// TwinCAT 3 PLC project PLC1
// ProgramVersion: 3.1.4023.0
// libraries:
//   Tc2_Standard, * (Beckhoff Automation GmbH)
//   Tc2_System, * (Beckhoff Automation GmbH)
//   Tc2_Utilities, * (Beckhoff Automation GmbH)
//   Tc3_Database, * (Beckhoff Automation GmbH)
//   Tc3_EventLogger, * (Beckhoff Automation GmbH)
//   Tc3_JsonXml, * (Beckhoff Automation GmbH)
//   Tc3_Module, * (Beckhoff Automation GmbH)
// project tree:
//   / DBTask.TcTTO
//   DUTs/ stData.TcDUT
//   GVLs/ GlobalData.TcGVL
//   POUs/ GetLocalData.TcPOU, GetLocalPlcEx.TcPOU, PostRemoteData.TcPOU, UpdateSync.TcPOU
// real-time tasks:
//   TASK PlcTask: cycle T#1ms, priority 20, ADS port 350
//   TASK PlcUpdateData: cycle T#100us, priority 21, ADS port 351
//   TASK DBTask: cycle T#100us, priority 22, ADS port 352

CONFIGURATION PLC1
    RESOURCE PLC ON TwinCAT3
        TASK DBTask(INTERVAL := T#100us, PRIORITY := 22);
        PROGRAM GetLocalData WITH DBTask : GetLocalData;
        PROGRAM PostRemoteData WITH DBTask : PostRemoteData;
        PROGRAM UpdateSync WITH DBTask : UpdateSync;
    END_RESOURCE
END_CONFIGURATION

// ---- DUTs/stData.TcDUT
TYPE stData :
STRUCT
	iId: LINT;
	bSync: BOOL;
	dtTimestamp: DT;
	rSpeed: LREAL;
	rPos: LREAL;
	bPulse: BOOL;
END_STRUCT
END_TYPE

// ---- GVLs/GlobalData.TcGVL
{attribute 'qualified_only'}
VAR_GLOBAL
	bRemotePosted: BOOL := FALSE;
	bLocalGot: BOOL:= FALSE;
	blocalUpdated: BOOL:= TRUE;
	bMeasure: BOOL;
	aReadStruct : stData;
END_VAR

// ---- POUs/GetLocalData.TcPOU
PROGRAM GetLocalData
VAR
	fbSqlDatabase : FB_SQLDatabaseEvt(sNetID := '', tTimeout := T#5S);
	fbSqlCommand : FB_SQLCommandEvt(sNetID := '', tTimeout := T#5S);
	fbSqlResult: FB_SQLResultEvt(sNetID:='', tTimeout := T#5S);
	myDBID: UDINT := 1;
	sTableName: STRING := 'Data';
	sCmd: STRING(1000);

	tcMessage1 : I_TcMessage;
	tcMessage2 : I_TcMessage;
	tcMessage3 : I_TcMessage;
	tcMessage4 : I_TcMessage;

	systime: GETSYSTEMTIME;
	currentTime: T_FILETIME;
	iId: LINT := 1;
	
	bFirstScan: BOOL := TRUE;
	bExecute: bool;
	fbTon: TON;
	bLapse: BOOL := FALSE;
	bRead: BOOL:= FALSE;
	
	temp: INT;
END_VAR

IF (bFirstScan) THEN
	IF fbSqlDatabase.Connect(myDBID) THEN
		bFirstScan := FALSE;
		IF fbSqlDatabase.bError THEN
			tcMessage1:= fbSqlDatabase.ipTcResult;
			bFirstScan := TRUE;
		END_IF
	END_IF
END_IF

fbTon(IN:= NOT fbTon.Q, PT:= T#100mS);
IF fbTon.Q THEN
	bExecute := TRUE;
END_IF

IF bExecute AND NOT bFirstScan AND GlobalData.blocalUpdated THEN
	GlobalData.bMeasure:= TRUE;
	CreateSelect();
		
	IF fbSqlDatabase.CreateCmd(ADR(fbSqlCommand)) THEN
		IF fbSqlDatabase.bError THEN
			tcMessage2:= fbSqlDatabase.ipTcResult;
		END_IF
	END_IF
		
	IF NOT bRead THEN 
		IF fbSQLCommand.ExecuteDataReturn(ADR(sCmd), LEN(sCmd), ADR(fbSqlResult)) THEN
			IF fbSQLCommand.bError THEN
				tcMessage3 := fbSQLCommand.ipTcResult;
			END_IF
			bRead:= TRUE;
		END_IF
	ELSE
		IF fbSqlResult.Read(0, 1, ADR(GlobalData.aReadStruct), SIZEOF(GlobalData.aReadStruct), FALSE, TRUE) THEN
			IF fbSqlResult.bError THEN
				tcMessage4:= fbSqlResult.ipTcResult;
			END_IF
			bRead:= FALSE;
			bExecute:= FALSE;
			IF GlobalData.aReadStruct.iId <> 0 THEN
				GlobalData.blocalUpdated:= FALSE;
				GlobalData.bLocalGot:= TRUE;
			END_IF
		END_IF
	END_IF
	
END_IF

ACTION CreateSelect:
sCmd := 'SELECT * FROM ';
sCmd := concat(sCmd, sTableName);
sCmd := concat(sCmd, ' WHERE Sync=0 LIMIT 1');
END_ACTION

END_PROGRAM

// ---- POUs/PostRemoteData.TcPOU
PROGRAM PostRemoteData
VAR
	//Query Builder for Document DB
	fbNoSqlQueryBuilder_DocumentDB: FB_NoSQLQueryBuilder_DocumentDB;
	InsertQueryOption: T_QueryOptionDocumentDB_Insert;
	sDocument: STRING (1000);
	sDBName: STRING := 'Datalog';

	//Document json writer
	fbJsonWriter: FB_JsonSaxWriter;
	
	//Query Execution
	fbNoSqlQuery: FB_NoSQLQueryEvt(sNetID:= '', tTimeout:= T#5S);
	myDBID: UDINT := 2;
	TcMessage: I_TcMessage;
END_VAR

IF GlobalData.bLocalGot THEN
	CreateQuery();
	CreateDocument();
	
	IF fbNoSqlQuery.Execute(hDBID:= myDBID, iNoSQLQueryBuilder:= fbNoSqlQueryBuilder_DocumentDB) THEN
		GlobalData.bLocalGot := FALSE;
		GlobalData.bRemotePosted := TRUE;
		IF fbNoSqlQuery.bError THEN
			TcMessage:= fbNoSqlQuery.ipTcResult;
			GlobalData.bLocalGot := TRUE;
			GlobalData.bRemotePosted := FALSE;
		END_IF
	END_IF
END_IF

ACTION CreateDocument:
fbJsonWriter.StartObject();
fbJsonWriter.AddKey('Timestamp');
fbJsonWriter.AddDateTime(GlobalData.aReadStruct.dtTimestamp);
fbJsonWriter.AddKey('Speed');
fbJsonWriter.AddLreal(GlobalData.aReadStruct.rSpeed);
fbJsonWriter.AddKey('Pos');
fbJsonWriter.AddLreal(GlobalData.aReadStruct.rPos);
fbJsonWriter.AddKey('Pulse');
fbJsonWriter.AddBool(GlobalData.aReadStruct.bPulse);
fbJsonWriter.EndObject();
sDocument := fbJsonWriter.GetDocument();
fbJsonWriter.ResetDocument();
END_ACTION

ACTION CreateQuery:
InsertQueryOption.pDocuments := ADR(sDocument);
InsertQueryOption.cbDocuments := SIZEOF(sDocument);

fbNoSqlQueryBuilder_DocumentDB.eQueryType := E_DocumentDbQueryType.InsertOne;
fbNoSqlQueryBuilder_DocumentDB.sCollectionName := sDBName;
fbNoSqlQueryBuilder_DocumentDB.pQueryOptions := ADR(InsertQueryOption);
fbNoSqlQueryBuilder_DocumentDB.cbQueryOptions := SIZEOF(InsertQueryOption);
END_ACTION

END_PROGRAM

// ---- POUs/UpdateSync.TcPOU
PROGRAM UpdateSync
VAR
	fbSqlDatabase : FB_SQLDatabaseEvt(sNetID := '', tTimeout := T#5S);
	fbSqlCommand : FB_SQLCommandEvt(sNetID := '', tTimeout := T#5S);
	myDBID: UDINT := 1;
	sTableName: STRING := 'Data';
	sCmd: STRING(1000);
	
	tcMessage1 : I_TcMessage;
	tcMessage2 : I_TcMessage;
	
	bFirstScan: BOOL := TRUE;
END_VAR

IF (bFirstScan) THEN
	IF fbSqlDatabase.Connect(myDBID) THEN
		bFirstScan := FALSE;
		IF fbSqlDatabase.bError THEN
			tcMessage1:= fbSqlDatabase.ipTcResult;
			bFirstScan := TRUE;
		END_IF
	END_IF
END_IF

IF GlobalData.bRemotePosted THEN
	CreateUpdate();
		
	IF fbSqlDatabase.CreateCmd(ADR(fbSqlCommand)) THEN
		IF fbSqlDatabase.bError THEN
			tcMessage1:= fbSqlDatabase.ipTcResult;
		END_IF
	END_IF
		
	IF fbSQLCommand.Execute(ADR(sCmd), LEN(sCmd)) THEN
		IF fbSQLCommand.bError THEN
			tcMessage2 := fbSQLCommand.ipTcResult;
		END_IF
		GlobalData.bRemotePosted := FALSE;
		GlobalData.blocalUpdated := TRUE;
		GlobalData.bMeasure := FALSE;
	END_IF
END_IF

ACTION CreateUpdate:
sCmd := 'UPDATE ';
sCmd := concat(sCmd, sTableName);
sCmd := concat(sCmd, ' SET Sync=');
sCmd := concat(sCmd, BOOL_TO_STRING(TRUE));
sCmd := concat(sCmd, ' WHERE Id=');
sCmd := concat(sCmd, LINT_TO_STRING(GlobalData.aReadStruct.iId));
END_ACTION

END_PROGRAM

// ---- POUs/GetLocalPlcEx.TcPOU
PROGRAM GetLocalPlcEx
VAR
	fbPLCDBRead : FB_PLCDBReadEvt (sNetID := '', tTimeout := T#5S);
	ColumnNames_read : ARRAY [0..4] OF STRING(50);
	myDBID: uint := 1;
	sMyTableName : T_MaxString:='Data';
	myRecordRead : stData;
	tcMessage_read : I_TcMessage;

	fbTon: TON;
	bRead: bool;
END_VAR

fbTon(IN:= NOT fbTon.Q, PT:= T#200MS);
IF fbTon.Q THEN
	bRead:= TRUE;
END_IF

IF bRead THEN
	ColumnNames_read[0] := 'ID';
	ColumnNames_read[1] := 'Timestamp';
	ColumnNames_read[2] := 'Speed';
	ColumnNames_read[3] := 'Pos';
	ColumnNames_read[4] := 'Pulse';
	
	IF fbPLCDBRead.ReadStruct(
		hDBID:= myDBID,
		sTableName:= sMyTableName,
		pColumnNames:= ADR(ColumnNames_read),
		cbColumnNames:= SIZEOF(ColumnNames_read),
		sOrderByColumn:= 'ID', 
		eOrderType:= E_OrderType.DESC, 
		nStartIndex:= 0, 
		nRecordCount:= 1, 
		pData:= ADR(myRecordRead), 
		cbData:= SIZEOF(myRecordRead)
	)
	THEN
		IF fbPLCDBRead.bError THEN
		tcMessage_read := fbPLCDBRead.ipTcResult;
		END_IF
		bRead:= FALSE;
	END_IF	
END_IF

END_PROGRAM
